Staubli VAL3: ack.pgx

public program ack(num x_nHeaderTime, num x_nElapsedTime)
begin

  // display time between valid trajectory point received and ACK sent

  gotoxy(scMonitor, 0,9)
  put(scMonitor, "recvMsgHeader:")
  gotoxy(scMonitor, 15,9)
  put(scMonitor, toString(".4", x_nHeaderTime))

  gotoxy(scMonitor, 0,10)
  put(scMonitor, "other states:")
  gotoxy(scMonitor, 15,10)
  put(scMonitor, toString(".4", x_nElapsedTime))

end
